FUNCTION_BLOCK FB_TelescopeParkedState EXTENDS FB_TelescopeState
VAR_INPUT
END_VAR
VAR_OUTPUT
END_VAR
VAR
	pMachine : POINTER TO FB_TelescopeMachine;
END_VAR

METHOD FB_init : BOOL
VAR_INPUT
	bInitRetains : BOOL; // if TRUE, the retain variables are initialized (warm start / cold start)
	bInCopyCode : BOOL;  // if TRUE, the instance afterwards gets moved into the copy code (online change)
	pMachine : POINTER TO FB_TelescopeMachine;
END_VAR
THIS^.pMachine := pMachine;
END_METHOD

METHOD Initialize : BOOL
VAR_INPUT
END_VAR
END_METHOD

END_FUNCTION_BLOCK

(* stored: Version 1.1.0.1, ProductVersion 3.1.4024.15
   POU FB_TelescopeParkedState: Id {fee317fb-bf48-4714-9d76-2e33fa60c6a5}, SpecialFunc None
   Method FB_init: Id {939ce836-b748-4327-8af4-fef7b1a3e467}
   Method Initialize: Id {4201b0a3-9d27-49e5-99b9-0daae87f0ec5} *)
